// TIA Portal V19 export
DATA_BLOCK "FlyingCarriage"   // DB135
// stored: InstanceOfName FlyingCarriage_FB, InstanceOfType FB
"FlyingCarriage_FB"
   // VAR_INPUT
   //    AreaInterface : "AreaInterface";
   //    ZSI : "udt_ZoneSafetyInterface";
   //    DSI : "udt_DeviceSafetyInterface";
   //    Drive { ExternalAccessible := 'False'; ExternalVisible := 'False'; ExternalWritable := 'False'} : "TAx_DriveInterface";
   //    CIn : "udt_FlyingCarriage_CIn";
   //    DataIn { ExternalAccessible := 'False'; ExternalVisible := 'False'; ExternalWritable := 'False'} : Struct
   //       Pb_Bkw : Bool;
   //       Pb_Fwd : Bool;
   //       Pb_Pos : Bool;
   //       Pb_Zero : Bool;
   //       Pb_PresetPos : Bool;
   //       Fbk_Fan : Bool;
   //    END_STRUCT;
   //    Config { ExternalAccessible := 'False'; ExternalVisible := 'False'; ExternalWritable := 'False'} : "udt_FlyingCarriage_Config";
   // END_VAR
   // VAR_OUTPUT
   //    MachineInterface : "MachineInterface";
   //    DataOut : Struct
   //       Fan : Bool;
   //       LP_ZeroOK : Bool;
   //    END_STRUCT;
   // END_VAR
   // VAR_IN_OUT
   //    TO_Carriage : TO_SynchronousAxis;
   //    TO_Master : TO_PositioningAxis;
   //    TO_ZeroChk : TO_MeasuringInput;
   //    Parameter : "udt_FlyingCarriage_Parameter";
   //    FsParameter : "udt_FsParameter";
   // END_VAR
   // VAR
   //    Warning : Struct
   //       NotAutReady : Bool;
   //       ZeroChkRequest : Bool;
   //       Axis : "TAx_Warnings";
   //    END_STRUCT;
   //    Alarm : Struct
   //       NotHomed : Bool;
   //       ZeroChkFailed : Bool;
   //       ZeroChk_NotCatched : Bool;
   //       ZeroChk_NotReleased : Bool;
   //       TargetPosition_OutOfRange : Bool;
   //       Axis : "TAx_Alarms";
   //       ZeroChk : "TMeasuring_Alarms";
   //       Fan : "MotorAlr";
   //    END_STRUCT;
   //    Diag : Struct
   //       Ax : "TO_Diagnostic";
   //       ZeroChk : "TO_Diagnostic";
   //    END_STRUCT;
   //    COut : Struct
   //       Infeed_ReqON : Bool;
   //       CtrlSafe : Bool;
   //       Ax_InOperation : Bool;
   //       Standstill : Bool;
   //       CheckNext_Minus : Bool;
   //       CheckNext_Plus : Bool;
   //       PositioningDone : Bool;
   //       InSynch : Bool;
   //       ActualTargetPosAx : LReal;
   //    END_STRUCT;
   //    HMI : Struct
   //       Pb_PresetPos : Bool;
   //       PresetPosValue : LReal;
   //       LastPositionDetect : LReal;
   //       ManPosTarget : LReal;
   //       PositionNorm : Real;
   //    END_STRUCT;
   //    Ax { S7_SetPoint := 'True'} : "FlyingShearAxis";
   //    MeasInp_ZeroChk { S7_SetPoint := 'True'} : "MeasuringInput";
   //    M_MotorFan : "Motor";
   //    tonDelayFanOff { S7_SetPoint := 'True'} : IEC_TIMER;
   //    tonDelayNoPendingCommands : IEC_TIMER;
   //    Sts : Struct
   //       IsStandstill : Bool;
   //       AlarmsPresence : Bool;
   //       WarningsPresence : Bool;
   //       DriveMessagesPresence : Bool;
   //       AxisMessagePresence : Bool;
   //       InOperatin : Bool;
   //       DriveParReadWriteDone : Bool;
   //       DriveMessagesReadDone : Bool;
   //       Gen_Condition : Bool;
   //       Bkw_Condition : Bool;
   //       Fwd_Condition : Bool;
   //       NoManCmd : Bool;
   //       Positioning_Condition : Bool;
   //       MotionRequestInNegativeDirection : Bool;
   //       MotionRequestInPositiveDirection : Bool;
   //       InPosition : Bool;
   //       AtHomePosition : Bool;
   //       Target_PosAx : LReal;
   //       MissingToTarget : LReal;
   //       ActualLimitMinus : LReal;
   //       ActualLimitPlus : LReal;
   //       ZeroChk_LastPositionDetect : LReal;
   //       ZeroChk_MeasInLastID : UInt;
   //    END_STRUCT;
   //    Ctrl : Struct
   //       RstAlarms : Bool;
   //       SafeMotion : Bool;
   //       StopDueDoorOpeningRequest : Bool;
   //       StopSafe : Bool;
   //       StopInPhase : Bool;
   //       StopProgrammed : Bool;
   //       StopAborting : Bool;
   //       ReadSLSParam : Bool;
   //       DriveParReadWrite_Exe : Bool;
   //       DriveMessageRead_Exe : Bool;
   //       Fan : Bool;
   //       Man_JogPosBkw : Bool;
   //       Man_JogPosFwd : Bool;
   //       Man_Pos : Bool;
   //       Man_Zero : Bool;
   //       Zero_Bkw : Bool;
   //       Zero_Fwd : Bool;
   //       Zero_Home : Bool;
   //       Man_Zero_Bkw : Bool;
   //       Man_Zero_Fwd : Bool;
   //       Man_Zero_Home : Bool;
   //       Man_PresetPosition : Bool;
   //       Aut_Zero : Bool;
   //       Aut_PosAbs : Bool;
   //       Aut_GearPos : Bool;
   //    END_STRUCT;
   //    AckRstAlarms : Bool;
   //    Pb_Bkw_PEAux : Bool;
   //    Pb_Fwd_PEAux : Bool;
   //    Pb_Pos_PEAux : Bool;
   //    Pb_Zero_PEAux : Bool;
   //    Pb_PresetPos_PEAux : Bool;
   //    ZeroChk_LastID : UInt;
   // END_VAR
BEGIN
END_DATA_BLOCK
